Universal Robots PolyScope program: letra_K.urp

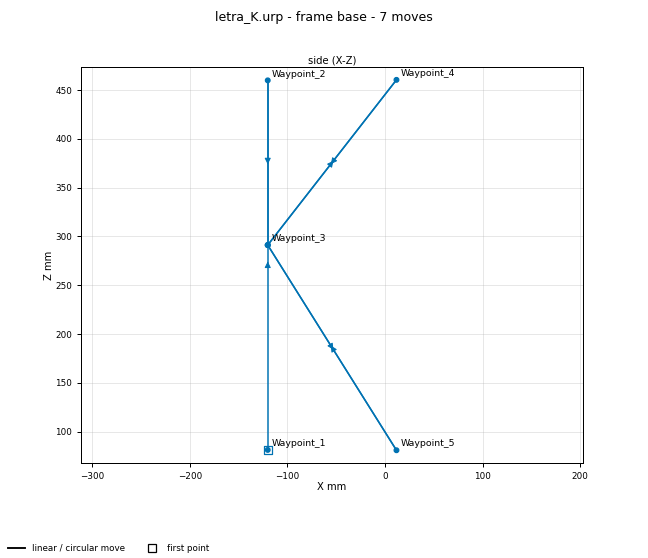
[picture p0: tool path of letra_K.urp in frame base, 7 of 7 moves have a stored position in this frame; points joined in program order, loops and branches not executed]
Program letra_K (installation=default directory=/ursim/programs createdIn=3.15.8.106339 lastSavedIn=3.15.8.106339 robotSerialNumber=2018359999)
Calibrated DH parameters: a=[0, -0.425, -0.39225, 0, 0, 0]; d=[0.089159, 0, 0, 0.10915, 0.09465, 0.0823]; alpha=[1.570796, 0, 0, 1.570796, -1.570796, 0]; deltaTheta=[0, 0, 0, 0, 0, 0]
Robot Program (runOnlyOnce=false)
  Popup Message (haltProgram=false message=Simulando letra K inputType=Text)
  MoveL speed 250 mm/s, acceleration 1200 mm/s^2 (useActiveTCP=true) feature=Base
    Waypoint Waypoint_1: TCP in base x=-120.113 y=-431.763 z=81.274 mm, rx=-0.0012 ry=3.1163 rz=0.0389 rad; joints [-91.713, -107.553, -129.299, -34.621, 91.393, -1.776] deg
    Waypoint Waypoint_2: TCP in base x=-120.113 y=-431.763 z=460 mm, rx=-0.0012 ry=3.1163 rz=0.0389 rad; joints [-91.713, -83.491, -91.645, -96.338, 91.393, -1.776] deg
    Waypoint Waypoint_3: TCP in base x=-120.113 y=-431.763 z=291.2 mm, rx=-0.0012 ry=3.1163 rz=0.0389 rad; joints [-91.713, -86.671, -113.859, -70.943, 91.393, -1.776] deg
    Waypoint Waypoint_4: TCP in base x=11.814 y=-437.802 z=460.521 mm, rx=-0.0012 ry=3.1163 rz=0.0389 rad; joints [-74.366, -81.998, -92.973, -96.02, 91.768, 15.574] deg
    Waypoint Waypoint_3: TCP in base x=-120.113 y=-431.763 z=291.2 mm, rx=-0.0012 ry=3.1163 rz=0.0389 rad; joints [-91.713, -86.671, -113.859, -70.943, 91.393, -1.776] deg
    Waypoint Waypoint_5: TCP in base x=11.814 y=-437.802 z=80.925 mm, rx=-0.0012 ry=3.1163 rz=0.0389 rad; joints [-74.366, -106.666, -131.019, -33.307, 91.768, 15.574] deg
    Waypoint Waypoint_3: TCP in base x=-120.113 y=-431.763 z=291.2 mm, rx=-0.0012 ry=3.1163 rz=0.0389 rad; joints [-91.713, -86.671, -113.859, -70.943, 91.393, -1.776] deg
